Fanuc KAREL source: V_CSAPI_GETVALUE.kl

PROGRAM T
%NOLOCKGROUP
VAR
 v0 : STRING[40]
 v1 : STRING[40]
 v2 : REAL
 v3 : INTEGER
BEGIN
 V_CSAPI_GETVALUE(v0, v1, v2, v3)
END T
